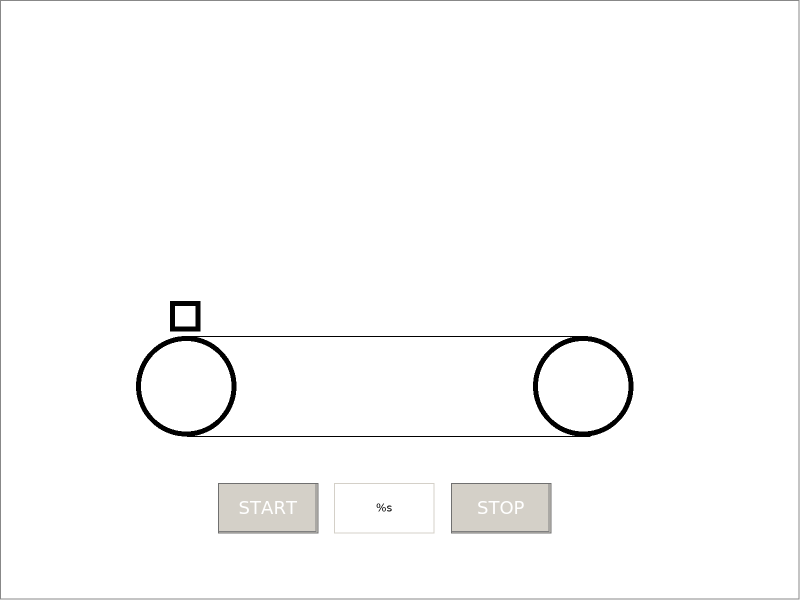
VISUALIZATION Visualization  // 800x600
    Group (136,336 497x101)
        Ellipse (0,0 100x100)
        Ellipse (397,0 100x100)
        Line (46,0) (449,0)
        Line (51,100) (454,100)
    Button (218,483 100x50), "START"
    Button (451,483 100x50), "STOP"
    Textfield (334,483 100x50), "%s"
    Rectangle (170,301 30x30)
END_VISUALIZATION

(* stored: Version 1.1.0.1, ProductVersion 3.1.4024.12
   Visu Visualization: Id {ec29af57-0a28-4724-ad79-761394bf8763} *)
